PROGRAM TEST
VAR
	//csvReader : FB_CsvReader;
END_VAR



//csvReader();

END_PROGRAM

(* stored: Version 1.1.0.1, ProductVersion 3.1.4022.18
   POU TEST: Id {f2edba56-12f7-486d-8838-64932ca9e828}, SpecialFunc None *)
